(* Logix 5000 project; controller cal1615 1756-L62 rev 20.19; software revision 20.05; part 46 of 81 *)
(* tags used below, declared in another part *)
   FAULT : BOOL;   // Fault AFI
   p01_recipe_active : recipe;   // Active Recipe
   p01r09_estop_ok : BOOL;   // System Modes Estop Dwell OK
   p01r09_pb_global_reset : BOOL;   // System Modes PB: Global Fault Reset
   p01r13_line_running : BOOL;   // System Line Start Sequence Line Running
   p01r13_state : DINT;   // System Line Start Sequence Sequencer Step
   p02_dint_from_hmi : hmi_dint;
   p02_real_from_hmi : hmi_real;   // MOP HMI Iface Real from HMI
   p20_di_acc_empty : BOOL;   // Letoff Digital Input Letoff Accumulator Empty Position
   p20r13_state : DINT;   // Letoff Accumulator State
   p21_ai_splice_platen_temp : REAL;   // Splice Press Analog Input Platen Temperature
   p21_ao_splice_platen_temp_cv : REAL;   // Splice Press Analog Output Platen Temp Command Value
   p21_di_platen_hi_temp_ok : BOOL;   // Splice Press Digital Input Platen High Temperature Ok
   p21_di_tc_bo : BOOL;   // Splice Press Digital Input Splice Platen Thermocouple Failure
   p21_do_close_exit_clamp_sv : BOOL;   // Splice Press Digital Output Close Exit Clamp
   p21_do_close_inlet_clamp_sv : BOOL;   // Splice Press Digital Output Close Inlet Clamp
   p21_do_enable_platen_heater : BOOL;   // Splice Press Digital Output Enable Platen Heater
   p21_pid_splice_press_temp : PID;   // Splice Press Temperature Control PID
   P21r01 : routine;
   p21r10 : routine;   // Splice Press Sequence
   p21r10_state : DINT;   // Splice Press Sequence State
   p21r10_status : DINT;   // Splice Press Sequence Status
   p21r10_timer_fault : TIMER[4];   // Splice Press Sequence Fault Delay
   p21r10_timer_warning : TIMER[4];   // Splice Press Sequence Warning Delay
   p21r16 : routine;   // Splice Press Temperature Control
   p21r16_pb_heater_off : BOOL;   // Splice Press Temperature Control PB: Heater Off
   p21r16_pb_heater_on : BOOL;   // Splice Press Temperature Control PB: Heater On
   p21r16_permissive_run : BOOL;   // Splice Press Temperature Control Permissive Run
   p21r16_pid_temp_cv : REAL;   // Splice Press Temperature Control PID Control Variable
   p21r16_pid_temp_pv : REAL;   // Splice Press Temperature Control PID Process Variable
   p21r16_pid_timer : TIMER;   // Splice Press Temperature Control PID Enable Timer
   p21r16_request_heat : BOOL;   // Splice Press Temperature Control Request Heat
   p21r16_timer_fault : TIMER[16];   // Splice Press Temperature Control Fault Delay
   p21r16_timer_warning : TIMER[16];   // Splice Press Temperature Control Warning Delay
   p22_di_close_nip_roll : BOOL;   // Tension Stand 1 Digital Input SS: Close Nip Roll
   p22_di_open_nip_roll : BOOL;   // Tension Stand 1 Digital Input SS: Open Nip Roll
   p22_dint_to_hmi : DINT[16];   // Tension Stand 1 Dint to HMI
   p22_do_close_nip_roll : BOOL;   // Tension Stand 1 Digital Output Close Tension Stand 1 Nip Roll
   p22r01 : routine;   // Tension Stand 1 Main
   p22r02 : routine;   // Tension Stand 1 Misc Control
   p22r02_fault_exists : BOOL;
   p22r02_nip_open : BOOL;
   p22r02_nip_open_dwell : TIMER;
   p22r02_request_system_run : BOOL;   // Tension Stand 1 Misc Control Request System Run
   p22r02_tension_dev_max : REAL;   // Winder A VFD
   p22r02_tension_dev_min : REAL;   // Tension Stand 1 VFD
   p22r02_timer_fault : TIMER[4];   // Tension Stand 1 Misc Control Fault Delay
   p22r02_timer_warning : TIMER[4];   // Tension Stand 1 Misc Control Warning Delay
   p22r02_unack_fault : BOOL;   // Impreg Pickup Roll Misc Control Unacknowledged Fault Exists
   p22r02_unack_warning : BOOL;   // Impreg Pickup Roll Misc Control Unacknowledged Warning Exists
   p22r02_warning_exists : BOOL;
   p22r03 : routine;   // Tension Stand 1 Input
   p22r04 : routine;   // Tension Stand 1 Output
   p22r05 : routine;   // Tension Stand 1 Dint to HMI
   p22r06 : routine;   // Tension Stand 1 Real to HMI
   p22r07 : routine;   // Tension Stand 1 Alarms
   p22r08 : routine;   // Tension Stand 1 Warnings
   p22r09 : routine;   // Tension Stand 1 Modes
   p22r10 : routine;   // Tension Stand 1 Speed Tension
   p22r11 : routine;   // Tension Stand 1 VFD
(* P21_Splice_Press, continued *)

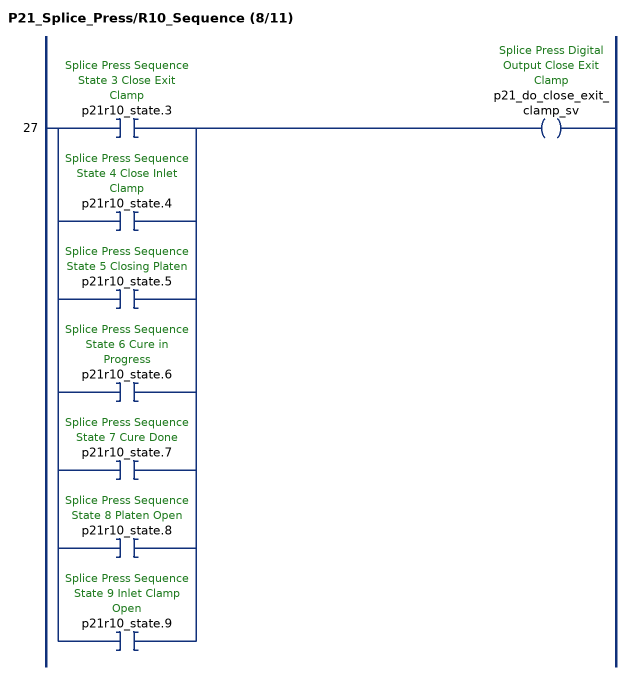
   [picture p880: P21_Splice_Press/R10_Sequence rungs 27-27]
   27: [XIC(p21r10_state.3) ,XIC(p21r10_state.4) ,XIC(p21r10_state.5) ,XIC(p21r10_state.6) ,XIC(p21r10_state.7) ,XIC(p21r10_state.8) ,XIC(p21r10_state.9) ]OTE(p21_do_close_exit_clamp_sv);
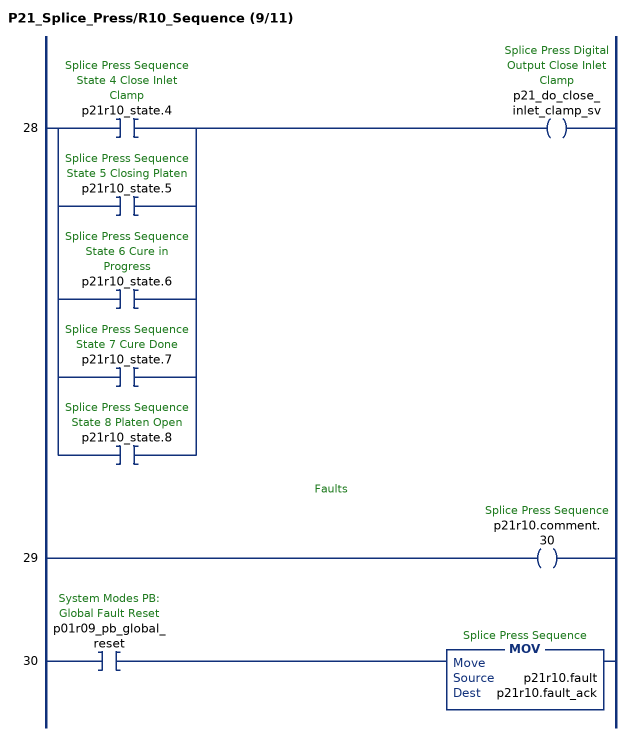
   28: [XIC(p21r10_state.4) ,XIC(p21r10_state.5) ,XIC(p21r10_state.6) ,XIC(p21r10_state.7) ,XIC(p21r10_state.8) ]OTE(p21_do_close_inlet_clamp_sv);
   // Faults
   29: OTE(p21r10.comment.30);
   30: XIC(p01r09_pb_global_reset)MOV(p21r10.fault,p21r10.fault_ack);
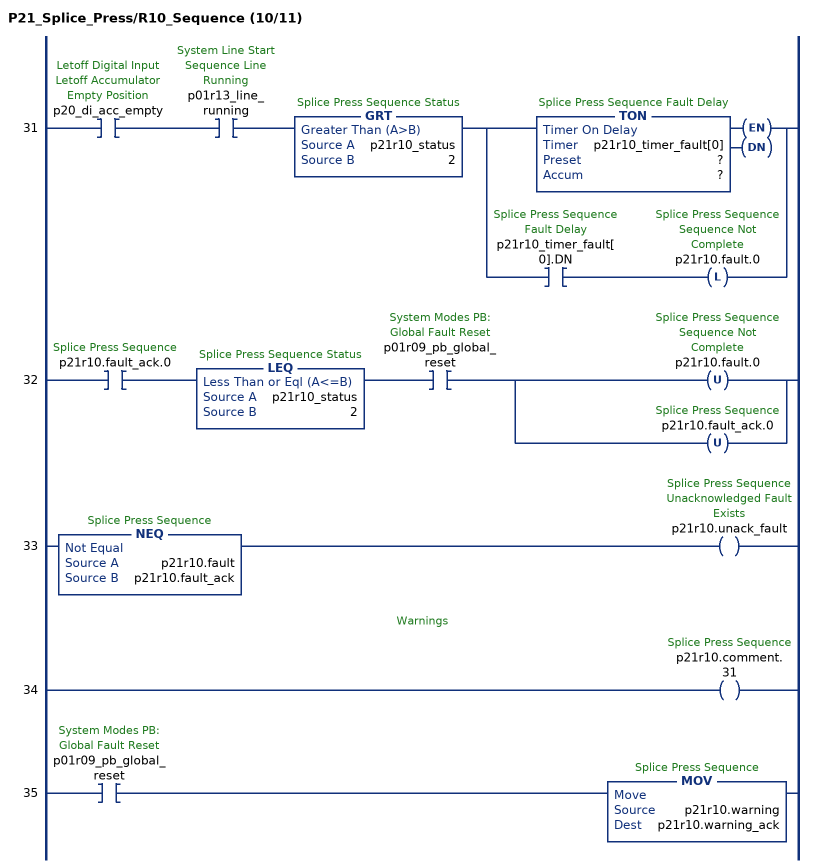
   31: XIC(p20_di_acc_empty)XIC(p01r13_line_running)GRT(p21r10_status,2)[TON(p21r10_timer_fault[0],?,?) ,XIC(p21r10_timer_fault[0].DN) OTL(p21r10.fault.0) ];
   32: XIC(p21r10.fault_ack.0)LEQ(p21r10_status,2)XIC(p01r09_pb_global_reset)[OTU(p21r10.fault.0) ,OTU(p21r10.fault_ack.0) ];
   33: NEQ(p21r10.fault,p21r10.fault_ack)OTE(p21r10.unack_fault);
   // Warnings
   34: OTE(p21r10.comment.31);
   35: XIC(p01r09_pb_global_reset)MOV(p21r10.warning,p21r10.warning_ack);
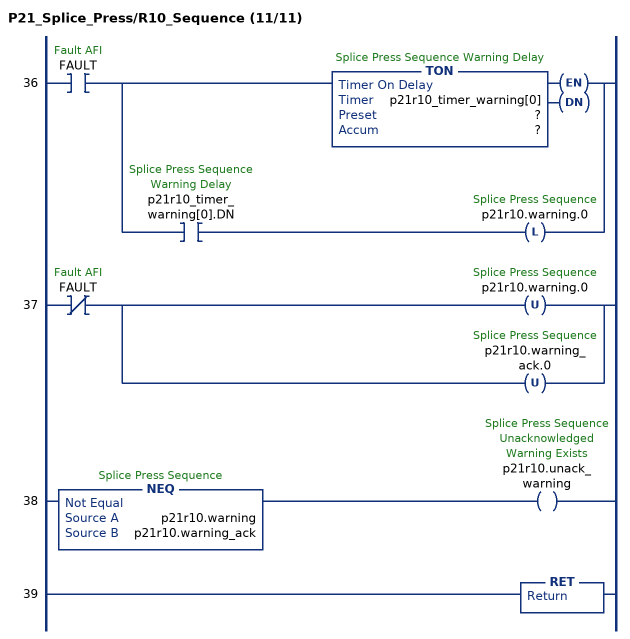
   36: XIC(FAULT)[TON(p21r10_timer_warning[0],?,?) ,XIC(p21r10_timer_warning[0].DN) OTL(p21r10.warning.0) ];
   37: XIO(FAULT)[OTU(p21r10.warning.0) ,OTU(p21r10.warning_ack.0) ];
   38: NEQ(p21r10.warning,p21r10.warning_ack)OTE(p21r10.unack_warning);
   39: RET();
END_ROUTINE

ROUTINE R16_Temperature_Control   (* ladder *)
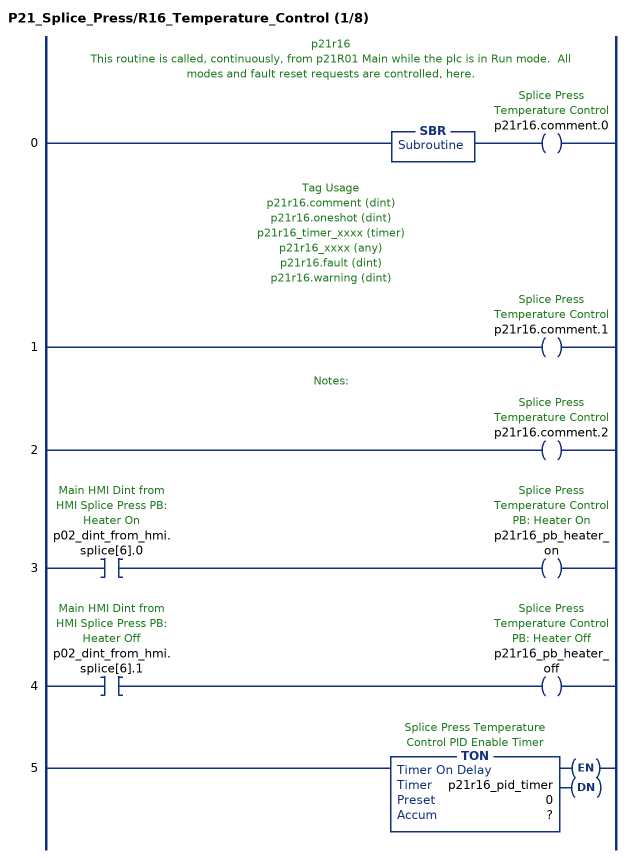
   // p21r16
   // This routine is called, continuously, from p21R01 Main while the plc is in Run mode.  All modes and fault reset requests are controlled, here.
   0: SBR()OTE(p21r16.comment.0);
   // Tag Usage
   // p21r16.comment (dint)
   // p21r16.oneshot (dint)
   // p21r16_timer_xxxx (timer)
   // p21r16_xxxx (any)
   // p21r16.fault (dint)
   // p21r16.warning (dint)
   1: OTE(p21r16.comment.1);
   // Notes:
   2: OTE(p21r16.comment.2);
   3: XIC(p02_dint_from_hmi.splice[6].0)OTE(p21r16_pb_heater_on);
   4: XIC(p02_dint_from_hmi.splice[6].1)OTE(p21r16_pb_heater_off);
   5: TON(p21r16_pid_timer,?,?);
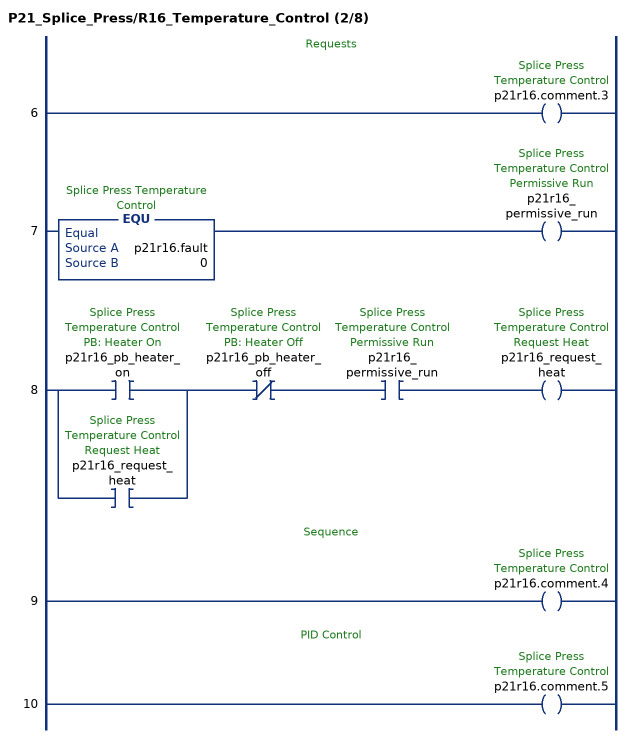
   // Requests
   6: OTE(p21r16.comment.3);
   7: EQU(p21r16.fault,0)OTE(p21r16_permissive_run);
   8: [XIC(p21r16_pb_heater_on) ,XIC(p21r16_request_heat) ]XIO(p21r16_pb_heater_off)XIC(p21r16_permissive_run)OTE(p21r16_request_heat);
   // Sequence
   9: OTE(p21r16.comment.4);
   // PID Control
   10: OTE(p21r16.comment.5);
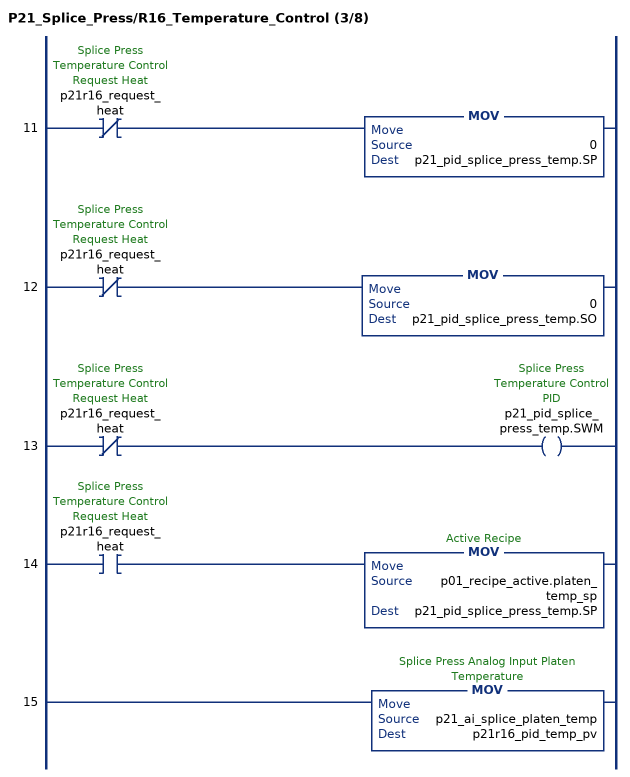
   11: XIO(p21r16_request_heat)MOV(0,p21_pid_splice_press_temp.SP);
   12: XIO(p21r16_request_heat)MOV(0,p21_pid_splice_press_temp.SO);
   13: XIO(p21r16_request_heat)OTE(p21_pid_splice_press_temp.SWM);
   14: XIC(p21r16_request_heat)MOV(p01_recipe_active.platen_temp_sp,p21_pid_splice_press_temp.SP);
   15: MOV(p21_ai_splice_platen_temp,p21r16_pid_temp_pv);
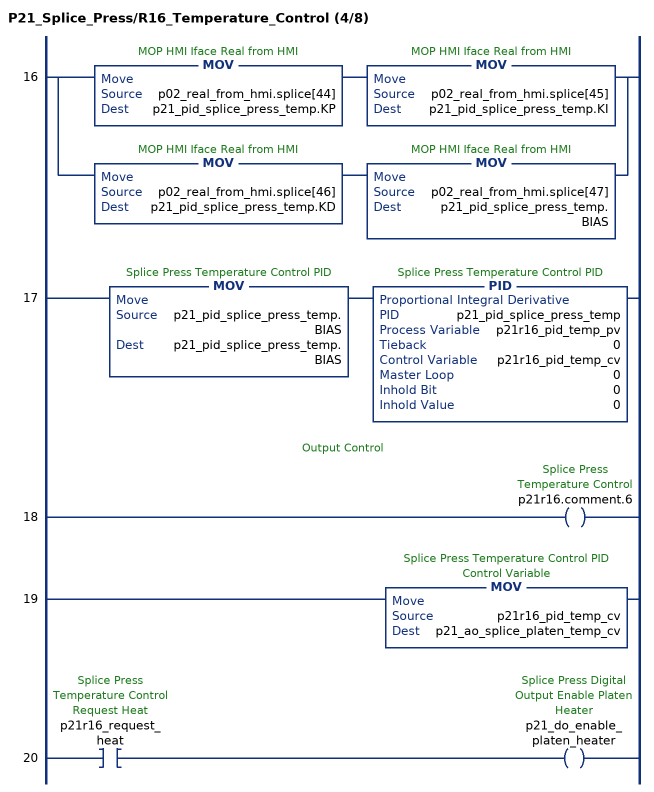
   16: [MOV(p02_real_from_hmi.splice[44],p21_pid_splice_press_temp.KP) MOV(p02_real_from_hmi.splice[45],p21_pid_splice_press_temp.KI) ,MOV(p02_real_from_hmi.splice[46],p21_pid_splice_press_temp.KD) MOV(p02_real_from_hmi.splice[47],p21_pid_splice_press_temp.BIAS) ];
   17: MOV(p21_pid_splice_press_temp.BIAS,p21_pid_splice_press_temp.BIAS)PID(p21_pid_splice_press_temp,p21r16_pid_temp_pv,0,p21r16_pid_temp_cv,0,0,0);
   // Output Control
   18: OTE(p21r16.comment.6);
   19: MOV(p21r16_pid_temp_cv,p21_ao_splice_platen_temp_cv);
   20: XIC(p21r16_request_heat)OTE(p21_do_enable_platen_heater);
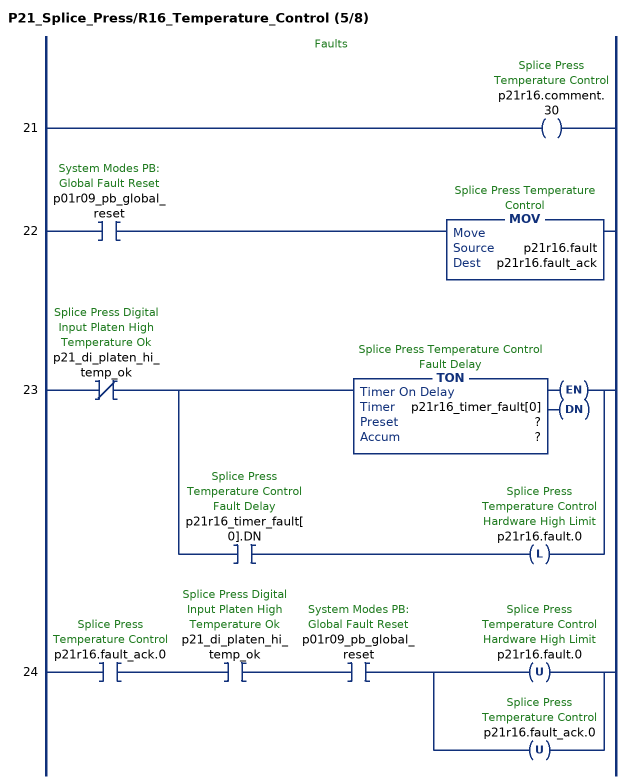
   // Faults
   21: OTE(p21r16.comment.30);
   22: XIC(p01r09_pb_global_reset)MOV(p21r16.fault,p21r16.fault_ack);
   23: XIO(p21_di_platen_hi_temp_ok)[TON(p21r16_timer_fault[0],?,?) ,XIC(p21r16_timer_fault[0].DN) OTL(p21r16.fault.0) ];
   24: XIC(p21r16.fault_ack.0)XIC(p21_di_platen_hi_temp_ok)XIC(p01r09_pb_global_reset)[OTU(p21r16.fault.0) ,OTU(p21r16.fault_ack.0) ];
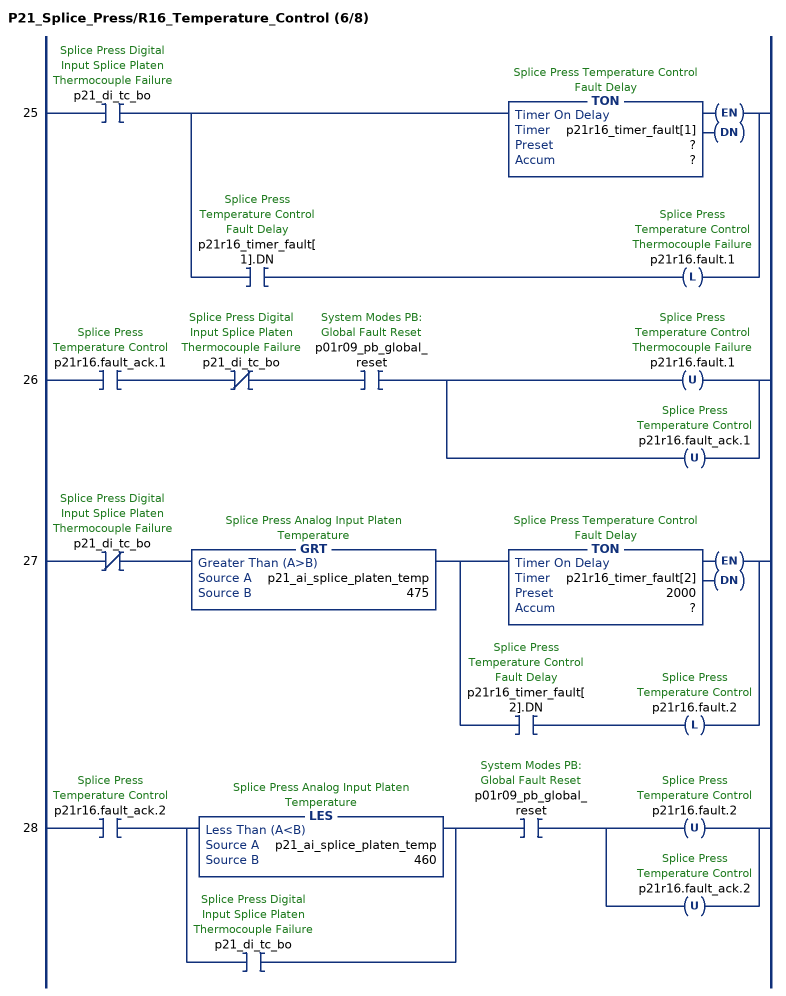
   25: XIC(p21_di_tc_bo)[TON(p21r16_timer_fault[1],?,?) ,XIC(p21r16_timer_fault[1].DN) OTL(p21r16.fault.1) ];
   26: XIC(p21r16.fault_ack.1)XIO(p21_di_tc_bo)XIC(p01r09_pb_global_reset)[OTU(p21r16.fault.1) ,OTU(p21r16.fault_ack.1) ];
   27: XIO(p21_di_tc_bo)GRT(p21_ai_splice_platen_temp,475)[TON(p21r16_timer_fault[2],?,?) ,XIC(p21r16_timer_fault[2].DN) OTL(p21r16.fault.2) ];
   28: XIC(p21r16.fault_ack.2)[LES(p21_ai_splice_platen_temp,460) ,XIC(p21_di_tc_bo) ]XIC(p01r09_pb_global_reset)[OTU(p21r16.fault.2) ,OTU(p21r16.fault_ack.2) ];
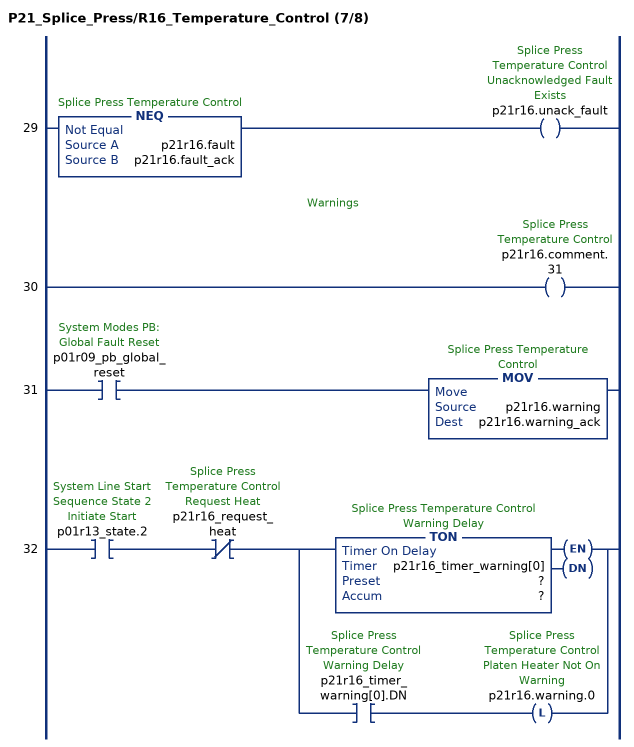
   29: NEQ(p21r16.fault,p21r16.fault_ack)OTE(p21r16.unack_fault);
   // Warnings
   30: OTE(p21r16.comment.31);
   31: XIC(p01r09_pb_global_reset)MOV(p21r16.warning,p21r16.warning_ack);
   32: XIC(p01r13_state.2)XIO(p21r16_request_heat)[TON(p21r16_timer_warning[0],?,?) ,XIC(p21r16_timer_warning[0].DN) OTL(p21r16.warning.0) ];
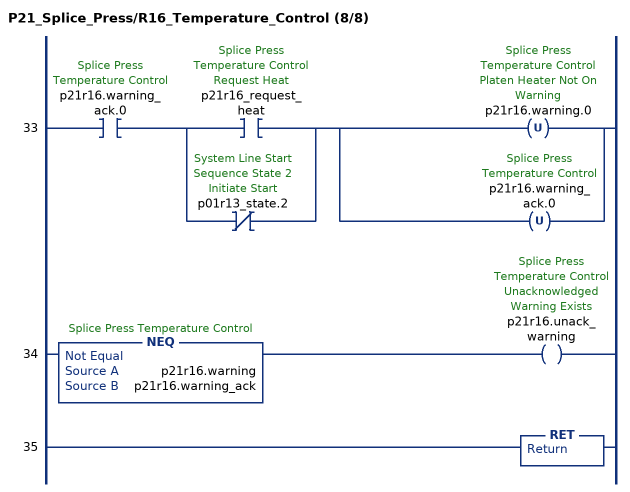
   33: XIC(p21r16.warning_ack.0)[XIC(p21r16_request_heat) ,XIO(p01r13_state.2) ][OTU(p21r16.warning.0) ,OTU(p21r16.warning_ack.0) ];
   34: NEQ(p21r16.warning,p21r16.warning_ack)OTE(p21r16.unack_warning);
   35: RET();
END_ROUTINE
END_PROGRAM

PROGRAM P22_Tension_Stand_1   (* main routine R01_Main *)

ROUTINE R01_Main   (* ladder *)
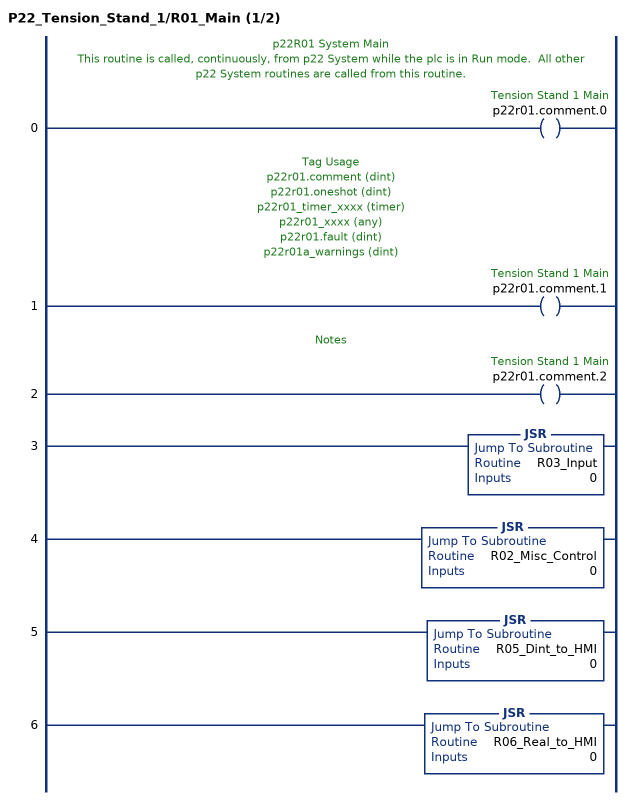
   // p22R01 System Main
   // This routine is called, continuously, from p22 System while the plc is in Run mode.  All other p22 System routines are called from this routine.
   0: OTE(p22r01.comment.0);
   // Tag Usage
   // p22r01.comment (dint)
   // p22r01.oneshot (dint)
   // p22r01_timer_xxxx (timer)
   // p22r01_xxxx (any)
   // p22r01.fault (dint)
   // p22r01a_warnings (dint)
   1: OTE(p22r01.comment.1);
   // Notes
   2: OTE(p22r01.comment.2);
   3: JSR(R03_Input,0);
   4: JSR(R02_Misc_Control,0);
   5: JSR(R05_Dint_to_HMI,0);
   6: JSR(R06_Real_to_HMI,0);
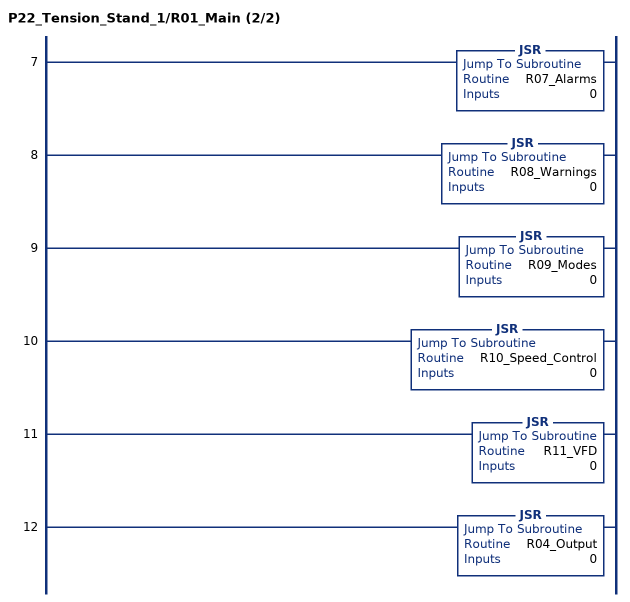
   7: JSR(R07_Alarms,0);
   8: JSR(R08_Warnings,0);
   9: JSR(R09_Modes,0);
   10: JSR(R10_Speed_Control,0);
   11: JSR(R11_VFD,0);
   12: JSR(R04_Output,0);
END_ROUTINE

ROUTINE R02_Misc_Control   (* ladder *)
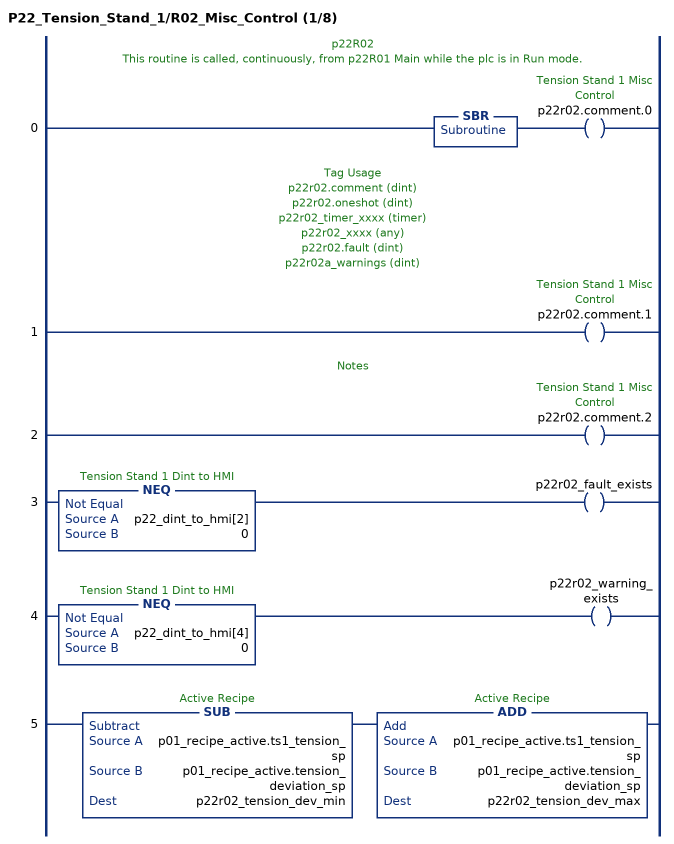
   // p22R02
   // This routine is called, continuously, from p22R01 Main while the plc is in Run mode.
   0: SBR()OTE(p22r02.comment.0);
   // Tag Usage
   // p22r02.comment (dint)
   // p22r02.oneshot (dint)
   // p22r02_timer_xxxx (timer)
   // p22r02_xxxx (any)
   // p22r02.fault (dint)
   // p22r02a_warnings (dint)
   1: OTE(p22r02.comment.1);
   // Notes
   2: OTE(p22r02.comment.2);
   3: NEQ(p22_dint_to_hmi[2],0)OTE(p22r02_fault_exists);
   4: NEQ(p22_dint_to_hmi[4],0)OTE(p22r02_warning_exists);
   5: SUB(p01_recipe_active.ts1_tension_sp,p01_recipe_active.tension_deviation_sp,p22r02_tension_dev_min)ADD(p01_recipe_active.ts1_tension_sp,p01_recipe_active.tension_deviation_sp,p22r02_tension_dev_max);
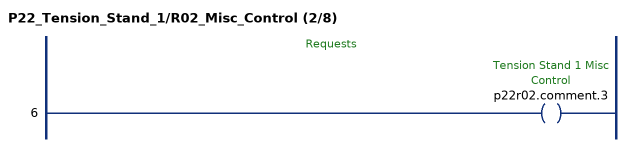
   // Requests
   6: OTE(p22r02.comment.3);
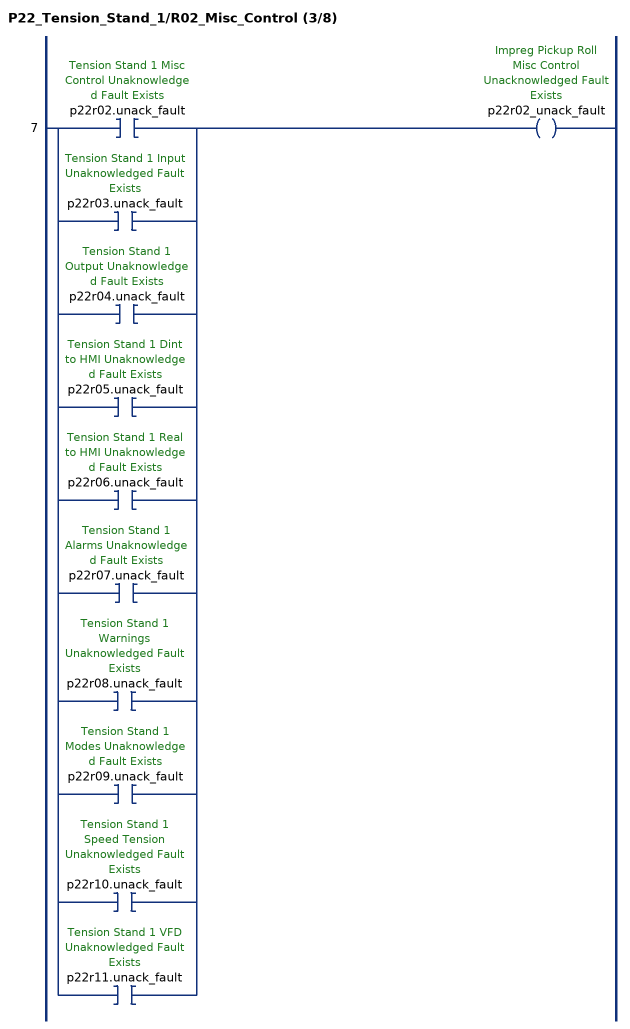
   7: [XIC(p22r02.unack_fault) ,XIC(p22r03.unack_fault) ,XIC(p22r04.unack_fault) ,XIC(p22r05.unack_fault) ,XIC(p22r06.unack_fault) ,XIC(p22r07.unack_fault) ,XIC(p22r08.unack_fault) ,XIC(p22r09.unack_fault) ,XIC(p22r10.unack_fault) ,XIC(p22r11.unack_fault) ]OTE(p22r02_unack_fault);
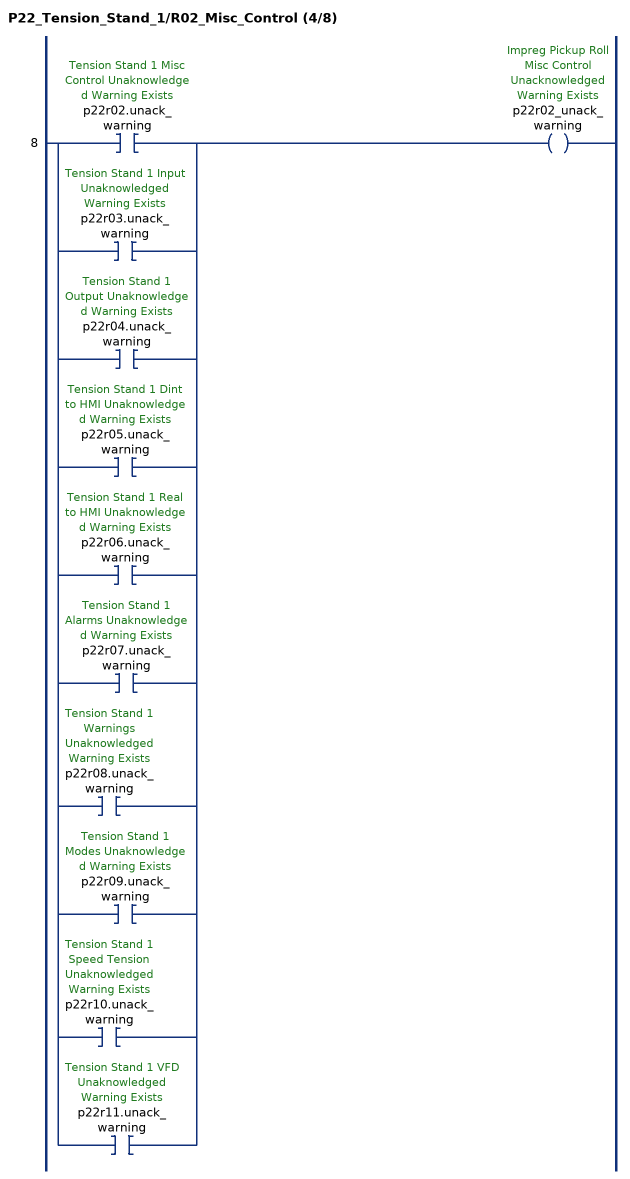
   8: [XIC(p22r02.unack_warning) ,XIC(p22r03.unack_warning) ,XIC(p22r04.unack_warning) ,XIC(p22r05.unack_warning) ,XIC(p22r06.unack_warning) ,XIC(p22r07.unack_warning) ,XIC(p22r08.unack_warning) ,XIC(p22r09.unack_warning) ,XIC(p22r10.unack_warning) ,XIC(p22r11.unack_warning) ]OTE(p22r02_unack_warning);
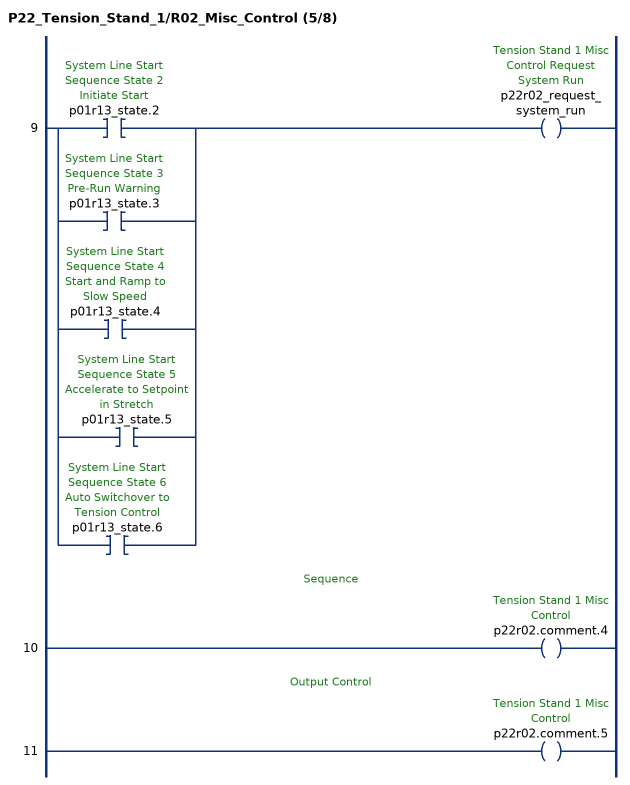
   9: [XIC(p01r13_state.2) ,XIC(p01r13_state.3) ,XIC(p01r13_state.4) ,XIC(p01r13_state.5) ,XIC(p01r13_state.6) ]OTE(p22r02_request_system_run);
   // Sequence
   10: OTE(p22r02.comment.4);
   // Output Control
   11: OTE(p22r02.comment.5);
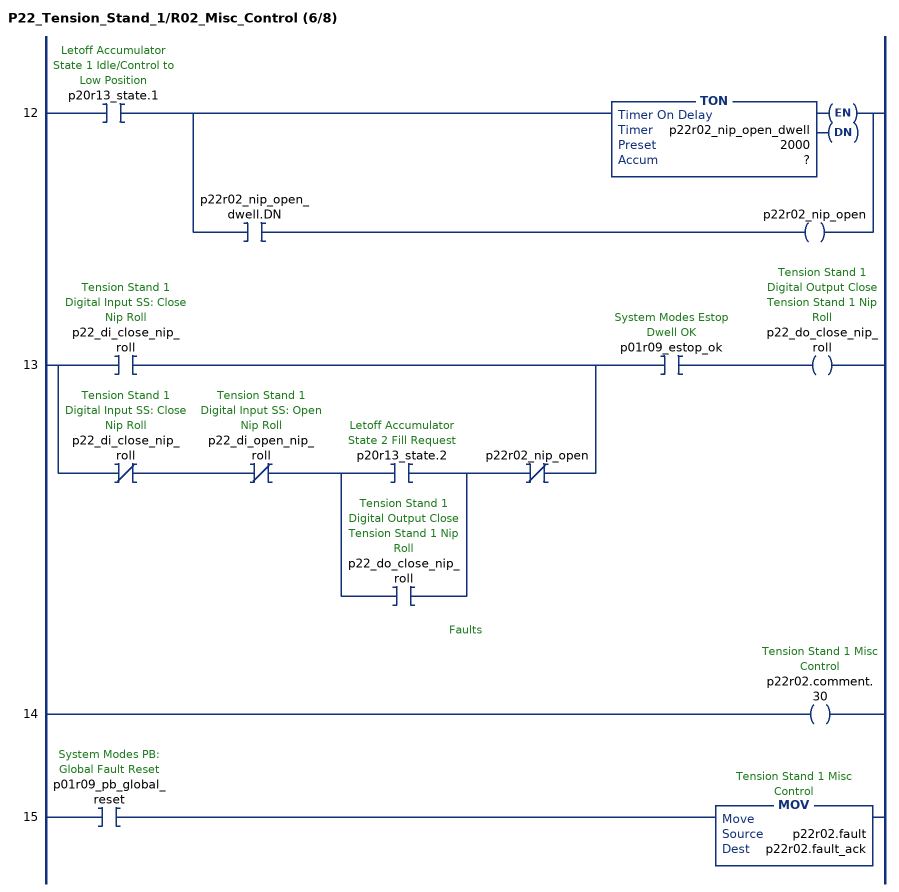
   12: XIC(p20r13_state.1)[TON(p22r02_nip_open_dwell,?,?) ,XIC(p22r02_nip_open_dwell.DN) OTE(p22r02_nip_open) ];
   13: [XIC(p22_di_close_nip_roll) ,XIO(p22_di_close_nip_roll) XIO(p22_di_open_nip_roll) [XIC(p20r13_state.2) ,XIC(p22_do_close_nip_roll) ] XIO(p22r02_nip_open) ]XIC(p01r09_estop_ok)OTE(p22_do_close_nip_roll);
   // Faults
   14: OTE(p22r02.comment.30);
   15: XIC(p01r09_pb_global_reset)MOV(p22r02.fault,p22r02.fault_ack);
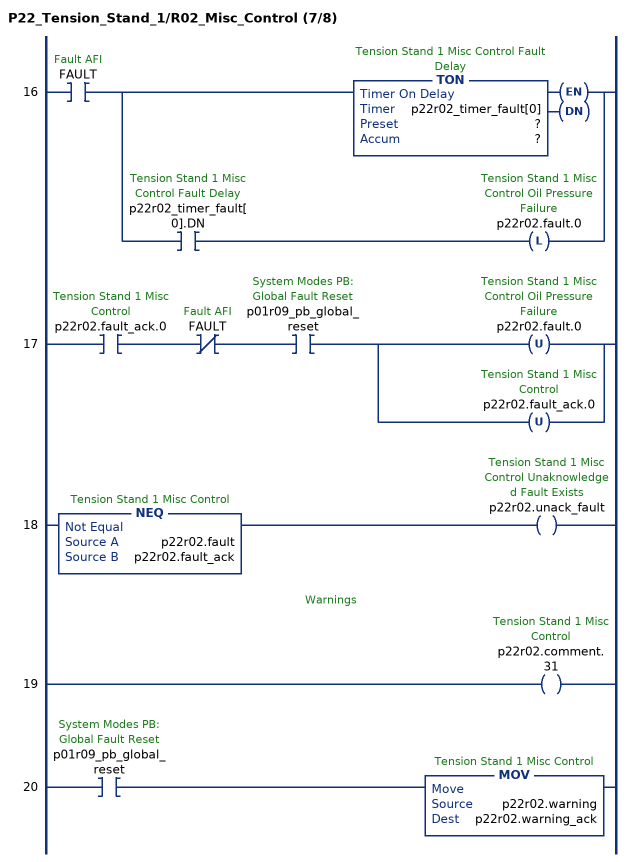
   16: XIC(FAULT)[TON(p22r02_timer_fault[0],?,?) ,XIC(p22r02_timer_fault[0].DN) OTL(p22r02.fault.0) ];
   17: XIC(p22r02.fault_ack.0)XIO(FAULT)XIC(p01r09_pb_global_reset)[OTU(p22r02.fault.0) ,OTU(p22r02.fault_ack.0) ];
   18: NEQ(p22r02.fault,p22r02.fault_ack)OTE(p22r02.unack_fault);
   // Warnings
   19: OTE(p22r02.comment.31);
   20: XIC(p01r09_pb_global_reset)MOV(p22r02.warning,p22r02.warning_ack);
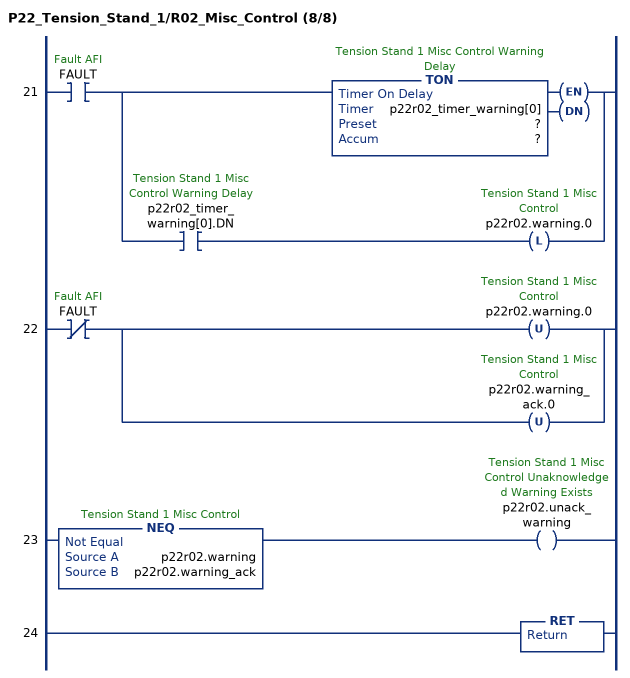
   21: XIC(FAULT)[TON(p22r02_timer_warning[0],?,?) ,XIC(p22r02_timer_warning[0].DN) OTL(p22r02.warning.0) ];
   22: XIO(FAULT)[OTU(p22r02.warning.0) ,OTU(p22r02.warning_ack.0) ];
   23: NEQ(p22r02.warning,p22r02.warning_ack)OTE(p22r02.unack_warning);
   24: RET();
END_ROUTINE
